TYPE typ_MotionManualMotion :
STRUCT
	MC_Jog				: MC_Jog;
END_STRUCT
END_TYPE

(* stored: Version 1.1.0.1, ProductVersion 3.1.4022.17
   DUT typ_MotionManualMotion: Id {b9a4fe59-5261-44da-9326-884764f5b028} *)
